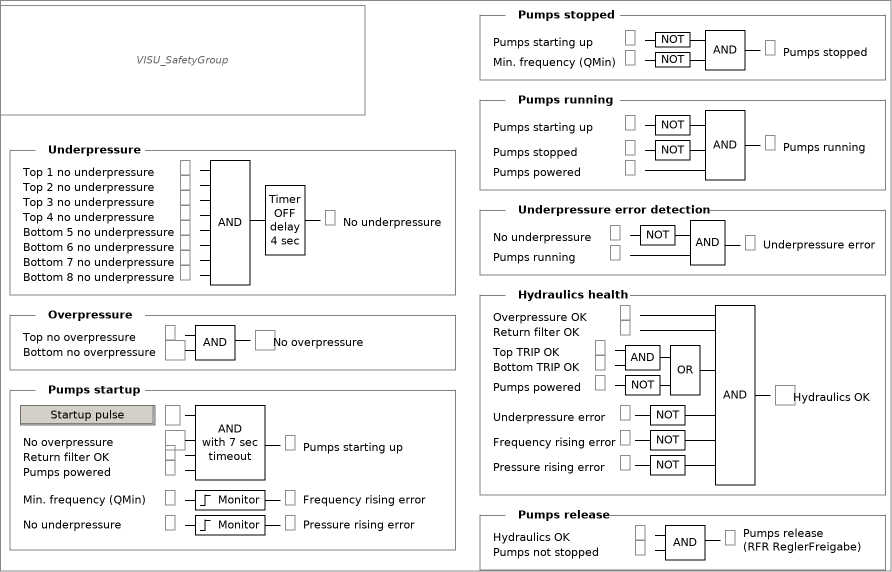
VISUALIZATION VISU_SafetyHydraulics  // 892x572
VAR_IN_OUT
	ref : SafetyHydraulics;
    widget : SafetyHydraulicsWidget;
END_VAR
    Polyline (630,295) (885,295) (885,495) (480,495) (480,295) (505,295)
    Polyline (710,210) (885,210) (885,275) (480,275) (480,210) (505,210)
    Polyline (145,390) (455,390) (455,550) (10,550) (10,390) (35,390)
    Polyline (145,150) (455,150) (455,295) (10,295) (10,150) (35,150)
    Button (20,405 135x20), "Startup pulse", input disabled if: ref.processes.startupPumps.statuses.enabledStatus.disabled
        OnMouseClick: execute { ref.processes.startupPumps.do_request := TRUE; }
    Frame (180,160 10x15)
        shows VISU_State_gray_green(state := ref.top1NoUnderpressure)
    Label (20,165 145x15), "Top 1 no underpressure"
    Label (20,180 135x15), "Top 2 no underpressure"
    Label (20,195 140x15), "Top 3 no underpressure"
    Label (20,210 140x15), "Top 4 no underpressure"
    Label (20,270 155x15), "Bottom 8 no underpressure"
    Label (20,225 155x15), "Bottom 5 no underpressure"
    Label (20,240 155x15), "Bottom 6 no underpressure"
    Label (20,255 155x15), "Bottom 7 no underpressure"
    Rectangle (210,160 40x125), "AND"
    Line (200,170) (210,170), colour toggle: ref.top1NoUnderpressure
    Rectangle (265,185 40x70), "Timer OFF delay 4 sec"
    Label (340,210 110x25), "No underpressure"
    Label (45,140 95x20), "Underpressure"
    Line (200,185) (210,185), colour toggle: ref.top2NoUnderpressure
    Line (200,200) (210,200), colour toggle: ref.top3NoUnderpressure
    Line (200,215) (210,215), colour toggle: ref.top4NoUnderpressure
    Line (200,230) (210,230), colour toggle: ref.bottom5NoUnderpressure
    Line (200,245) (210,245), colour toggle: ref.bottom6NoUnderpressure
    Line (200,260) (210,260), colour toggle: ref.bottom7NoUnderpressure
    Line (200,275) (210,275), colour toggle: ref.bottom8NoUnderpressure
    Line (250,220) (265,220), colour toggle: ref.noUnderpressureNoDelay
    Line (305,220) (320,220), colour toggle: ref.noUnderpressure
    Polyline (145,315) (455,315) (455,370) (10,370) (10,315) (35,315)
    Frame (255,330 20x20)
        shows VISU_State_red_green(state := ref.noOverpressure)
    Frame (165,325 10x15)
        shows VISU_State_red_green(state := ref.topNoOverpressure)
    Label (20,330 140x15), "Top no overpressure"
    Label (20,345 140x15), "Bottom no overpressure"
    Frame (165,340 20x20)
        shows VISU_State_red_green(state := ref.bottomNoOverpressure)
    Rectangle (195,325 40x35), "AND"
    Line (185,335) (195,335), colour toggle: ref.topNoOverpressure
    Label (270,330 105x25), "No overpressure"
    Label (45,305 95x20), "Overpressure"
    Line (185,350) (195,350), colour toggle: ref.bottomNoOverpressure
    Line (235,340) (250,340), colour toggle: ref.noOverpressure
    Frame (285,435 10x15)
        shows VISU_State_gray_green(state := ref.pumpsStartingUp)
    Frame (165,405 15x20)
        shows VISU_State_gray_green(state := ref.restartPumpsOutput)
    Label (20,435 110x15), "No overpressure"
    Frame (165,430 20x20)
        shows VISU_State_red_green(state := ref.noOverpressure)
    Rectangle (195,405 70x75), "AND with 7 sec timeout"
    Line (185,415) (195,415), colour toggle: ref.restartPumpsOutput
    Label (300,435 115x25), "Pumps starting up"
    Label (45,380 95x20), "Pumps startup"
    Line (185,440) (195,440), colour toggle: ref.noOverpressure
    Line (265,445) (280,445), colour toggle: ref.pumpsStartingUp
    Label (20,450 100x15), "Return filter OK"
    Frame (165,445 10x15)
        shows VISU_State_green_red(state := ref.returnFilterOverpressure)
    Line (185,455) (195,455), colour toggle: ref.returnFilterOverpressure
    Frame (165,490 10x15)
        shows VISU_State_gray_green(state := ref.pumpsMinFrequency)
    Rectangle (195,490 70x20)
    Frame (285,490 10x15)
        shows VISU_State_gray_red(state := ref.pumpsFrequencyNotRising)
    Label (300,490 125x20), "Frequency rising error"
    Line (265,500) (280,500), colour toggle: ref.pumpsFrequencyNotRising
    Label (20,490 140x20), "Min. frequency (QMin)"
    Rectangle (195,515 70x20)
    Label (300,515 125x20), "Pressure rising error"
    Label (20,515 125x20), "No underpressure"
    Polyline (620,15) (885,15) (885,80) (480,80) (480,15) (505,15)
    Frame (765,40 10x15)
        shows VISU_State_gray_green(state := ref.pumpsStopped)
    Label (490,35 140x15), "Pumps starting up"
    Label (490,55 140x15), "Min. frequency (QMin)"
    Frame (625,50 10x15)
        shows VISU_State_gray_green(state := ref.pumpsMinFrequency)
    Rectangle (705,30 40x40), "AND"
    Line (690,40) (705,40), colour toggle: ref.pumpsStartingUp
    Label (780,40 90x25), "Pumps stopped"
    Label (515,5 160x20), "Pumps stopped"
    Line (745,50) (760,50), colour toggle: ref.pumpsStopped
    Frame (775,385 20x20)
        shows VISU_State_red_green(state := ref.allOK)
    Label (490,230 105x15), "No underpressure"
    Label (490,250 140x15), "Pumps running"
    Frame (610,245 10x15)
        shows VISU_State_gray_green(state := ref.pumpsRunning)
    Rectangle (690,220 35x45), "AND"
    Label (790,385 100x25), "Hydraulics OK"
    Line (755,395) (770,395), colour toggle: ref.allOK
    Rectangle (715,305 40x180), "AND"
    Label (490,310 135x15), "Overpressure OK"
    Frame (620,305 10x15)
        shows VISU_State_red_green(state := ref.noOverpressure)
    Line (640,315) (715,315), colour toggle: ref.noOverpressure
    Label (490,325 135x15), "Return filter OK"
    Label (490,345 135x15), "Top TRIP OK"
    Frame (595,340 10x15)
        shows VISU_State_red_green(state := ref.topTripOK)
    Line (615,350) (625,350), colour toggle: ref.topTripOK
    Label (490,360 135x15), "Bottom TRIP OK"
    Frame (595,355 10x15)
        shows VISU_State_red_green(state := ref.bottomTripOK)
    Line (615,365) (625,365), colour toggle: ref.bottomTripOK
    Label (515,285 140x20), "Hydraulics health"
    Polyline (610,515) (885,515) (885,570) (480,570) (480,515) (505,515)
    Frame (725,530 10x15)
        shows VISU_State_gray_green(state := ref.pumpsRelease)
    Frame (635,525 10x15)
        shows VISU_State_red_green(state := ref.allOK)
    Label (490,530 140x15), "Hydraulics OK"
    Label (490,545 140x15), "Pumps not stopped"
    Frame (635,540 10x15)
        shows VISU_State_green_gray(state := ref.pumpsStopped)
    Rectangle (665,525 40x35), "AND"
    Line (655,535) (665,535), colour toggle: ref.allOK
    Label (740,520 130x40), "Pumps release (RFR ReglerFreigabe)"
    Label (515,505 95x20), "Pumps release"
    Line (655,550) (665,550), colour toggle: ref.pumpsStopped
    Line (705,540) (720,540), colour toggle: ref.pumpsRelease
    Label (215,515 45x20), "Monitor"
    Label (215,490 45x20), "Monitor"
    Polyline (200,530) (205,530) (205,520) (210,520)
    Frame (0,5 365x110)
        shows VISU_SafetyGroup(statusWidget := widget.actualStatus, comError := ref.groupComError, fbError := ref.groupFbError, outError := ref.groupOutError, reset := ref.processes.reset)
    Line (185,500) (195,500), colour toggle: ref.pumpsMinFrequency
    Frame (285,515 10x15)
        shows VISU_State_gray_red(state := ref.pressureNotRising)
    Line (265,525) (280,525), colour toggle: ref.pressureNotRising
    Frame (620,320 10x15)
        shows VISU_State_green_red(state := ref.returnFilterOverpressure)
    Line (640,330) (715,330), colour toggle: ref.returnFilterOverpressure
    Line (685,440) (715,440), colour toggle: ref.pumpsFrequencyNotRising
    Line (685,465) (715,465), colour toggle: ref.pressureNotRising
    Label (490,435 140x15), "Frequency rising error"
    Label (490,460 140x15), "Pressure rising error"
    Frame (180,175 10x15)
        shows VISU_State_gray_green(state := ref.top2NoUnderpressure)
    Frame (180,190 10x15)
        shows VISU_State_gray_green(state := ref.top3NoUnderpressure)
    Frame (180,205 10x15)
        shows VISU_State_gray_green(state := ref.top4NoUnderpressure)
    Frame (180,220 10x15)
        shows VISU_State_gray_green(state := ref.bottom5NoUnderpressure)
    Frame (180,235 10x15)
        shows VISU_State_gray_green(state := ref.bottom6NoUnderpressure)
    Frame (180,250 10x15)
        shows VISU_State_gray_green(state := ref.bottom7NoUnderpressure)
    Frame (180,265 10x15)
        shows VISU_State_gray_green(state := ref.bottom8NoUnderpressure)
    Frame (325,210 10x15)
        shows VISU_State_gray_green(state := ref.noUnderpressure)
    Frame (165,515 10x15)
        shows VISU_State_gray_green(state := ref.noUnderpressure)
    Line (185,525) (195,525), colour toggle: ref.noUnderpressure
    Line (685,415) (715,415), colour toggle: ref.underpressureError
    Label (490,410 140x15), "Underpressure error"
    Label (515,200 195x20), "Underpressure error detection"
    Frame (610,225 10x15)
        shows VISU_State_gray_green(state := ref.noUnderpressure)
    Rectangle (640,225 35x20), "NOT"
    Line (725,245) (740,245), colour toggle: ref.underpressureError
    Label (760,235 125x20), "Underpressure error"
    Frame (745,235 10x15)
        shows VISU_State_gray_red(state := ref.underpressureError)
    Polyline (620,100) (885,100) (885,190) (480,190) (480,100) (505,100)
    Frame (765,135 10x15)
        shows VISU_State_gray_green(state := ref.pumpsRunning)
    Label (490,120 140x15), "Pumps starting up"
    Label (490,145 140x15), "Pumps stopped"
    Frame (625,140 10x15)
        shows VISU_State_gray_green(state := ref.pumpsStopped)
    Rectangle (705,110 40x70), "AND"
    Label (780,135 90x25), "Pumps running"
    Label (515,90 160x20), "Pumps running"
    Line (645,150) (655,150), colour toggle: ref.pumpsStopped
    Line (745,145) (760,145), colour toggle: ref.pumpsRunning
    Rectangle (655,32 35x15), "NOT"
    Line (645,40) (655,40), colour toggle: ref.pumpsStartingUp
    Rectangle (655,115 35x20), "NOT"
    Rectangle (655,140 35x20), "NOT"
    Frame (625,30 10x15)
        shows VISU_State_gray_green(state := ref.pumpsStartingUp)
    Frame (625,115 10x15)
        shows VISU_State_gray_green(state := ref.pumpsStartingUp)
    Line (690,125) (705,125), colour toggle: ref.pumpsStartingUp
    Line (645,125) (655,125), colour toggle: ref.pumpsStopped
    Line (690,150) (705,150), colour toggle: ref.pumpsStopped
    Line (630,235) (640,235), colour toggle: ref.noUnderpressure
    Line (630,255) (690,255), colour toggle: ref.pumpsRunning
    Line (675,235) (690,235), colour toggle: ref.noUnderpressure
    Rectangle (650,405 35x20), "NOT"
    Rectangle (650,430 35x20), "NOT"
    Rectangle (650,455 35x20), "NOT"
    Line (635,415) (650,415), colour toggle: ref.underpressureError
    Frame (620,405 10x15)
        shows VISU_State_gray_red(state := ref.underpressureError)
    Frame (620,430 10x15)
        shows VISU_State_gray_red(state := ref.pumpsFrequencyNotRising)
    Frame (620,455 10x15)
        shows VISU_State_gray_red(state := ref.pressureNotRising)
    Line (635,465) (650,465), colour toggle: ref.pressureNotRising
    Line (635,440) (650,440), colour toggle: ref.pumpsFrequencyNotRising
    Polyline (200,505) (205,505) (205,495) (210,495)
    Line (645,60) (655,60), colour toggle: ref.pumpsMinFrequency
    Line (690,60) (705,60), colour toggle: ref.pumpsMinFrequency
    Rectangle (655,52 35x15), "NOT"
    Rectangle (625,345 35x25), "AND"
    Frame (595,375 10x15)
        shows VISU_State_gray_green(state := ref.pumpsPowered)
    Line (615,385) (625,385), colour toggle: ref.pumpsPowered
    Label (490,380 100x15), "Pumps powered"
    Rectangle (625,375 35x20), "NOT"
    Line (660,385) (675,385), colour toggle: ref.pumpsPowered
    Rectangle (670,345 30x50), "OR"
    Line (700,370) (715,370), colour toggle: ref.pumpsPowered OR (ref.topTripOK AND ref.bottomTripOK)
    Label (490,165 140x15), "Pumps powered"
    Frame (625,160 10x15)
        shows VISU_State_gray_green(state := ref.pumpsPowered)
    Line (645,170) (705,170), colour toggle: ref.pumpsPowered
    Line (660,357) (670,357), colour toggle: ref.topTripOK AND ref.bottomTripOK
    Frame (165,460 10x15)
        shows VISU_State_gray_green(state := ref.pumpsPowered)
    Line (185,470) (195,470), colour toggle: ref.pumpsPowered
    Label (20,465 100x15), "Pumps powered"
END_VISUALIZATION

(* stored: Version 1.1.0.1, ProductVersion 3.1.4019.2
   Visu VISU_SafetyHydraulics: Id {2a8c80dd-c7fd-4c6a-8169-22c4fe6bdd0a} *)
